Fanuc KAREL source: kb00034.KL

-- PROVISIONAL review KL for V940-1; original PC SHA256 c25f7c17c73512dcf3a1b786857e99abbf6a20790b8bf78608b49ea0ad8b607c
-- Incomplete behavior may be omitted. Consult companion uncertainty JSON. Do not deploy.
PROGRAM KB00034
%NOLOCKGROUP
BEGIN
  -- V9_ZERO_TABLE_METADATA_HINT layout=0002_ascii; no indexed target words; source/name/runtime held
  -- UNRESOLVED_PC offsets 5-14; opcodes 3F,75
  -- UNRESOLVED_PC offsets 19-37; opcodes 27,22,22,2A,31
  -- UNRESOLVED_PC offsets 42-46; opcodes 7F
END KB00034
